// TIA Portal V20 export
FUNCTION_BLOCK "FB_Temperature"   // FB490, SCL
{ S7_Optimized_Access := 'TRUE' }
// stored: AutoNumber false, MemoryReserve 100, SetENOAutomatically false
   VAR
      sPIDRestart : Bool;
      sPIDHoldI : Bool;
      sXAxisWarning : Real := 50.0;
      sPIDClimOut : Real;
      sP : Real := -100.0;
      sI : Time := T#10D;
      sD : Time := T#12S;
      sTimeOutFlowChiller : TON_TIME;
      sTimeOutLevelChiller { S7_SetPoint := 'True'} : TON_TIME;
      sTimeOutChillerGood : TON_TIME;
      sTimeOutCooling : TON_TIME;
      sTemperature_X_PT1000 { S7_SetPoint := 'True'} : "FB_AnalogInputThreshold";
      sTemperature_Y_PT1000 { S7_SetPoint := 'True'} : "FB_AnalogInputThreshold";
      sAmbiantTemperature { S7_SetPoint := 'True'} : "FB_AnalogInputThreshold";
      sMachineTemperature { S7_SetPoint := 'True'} : "FB_AnalogInputThreshold";
      sCabinetTemperatureMeasure { S7_SetPoint := 'True'} : "FB_AnalogInputThreshold";
      sColdWaterTemperatureInput { S7_SetPoint := 'True'} : "FB_AnalogInputThreshold";
      sColdWaterTemperatureOutput { S7_SetPoint := 'True'} : "FB_AnalogInputThreshold";
      sTemperatureCooling { S7_SetPoint := 'True'} : "FB_AnalogInputThreshold";
   END_VAR
   VAR_TEMP
      tSetPointCheck : Real;
      tDataAction : "AnalogInAction_DT";
   END_VAR
   VAR CONSTANT
      ALARM_PTC : Real := 110.0;
      TIME_OUT_COOLING : Time := T#5S;
   END_VAR
BEGIN
   REGION Description header 
       //==================================================================================
       // POSALUX Swiss SA / (C) Copyright 2024
       //----------------------------------------------------------------------------------
       // Title: Temperatures management
       // Comment/Function: 
       //
       // Author: Gowsigan SRITHARAN
       // Engineering: TIA Portal v17
       //----------------------------------------------------------------------------------
       // Change log table:
       // Version  | Date     | Expert in charge | Changes applied
       // ---------|----------|------------------|------------------------------------
       // 00.00.01 | 20241120 | GSR              | First released version
       // ==================================================================================
   END_REGION

   REGION Ambiant temperature (externe)  
       #sAmbiantTemperature(iActualValue := "DB_AnalogInputs".sAmbiantTemperature.sSWRealValue,
                            iStartDelay := TRUE,
                            ioAlarmMin := "LBP_AlarmMsgs".UserA[06].A70UUxx[04],
                            ioWarningMin := "LBP_AlarmMsgs".UserA[07].A70UUxx[04],
                            ioWarningMax := "LBP_AlarmMsgs".UserA[07].A70UUxx[05],
                            ioAlarmMax := "LBP_AlarmMsgs".UserA[06].A70UUxx[05],
                            oDataAction => "DB_AnalogInputAction".Ambiant_Temperature,
                            iDataPLC := "DB_AnalogInputDataPLC".Ambiant_Temperature,
                            iDataHMI := "DB_AnalogInputDataHMI".Ambiant_Temperature);
   END_REGION

   REGION Water input  
       #sColdWaterTemperatureInput(iActualValue := "DB_AnalogInputs".sCold_WaterTemperatureInput.sSWRealValue,
                                   iStartDelay := TRUE,
                                   ioAlarmMin := "LBP_AlarmMsgs".UserA[06].A70UUxx[08],
                                   ioWarningMin := "LBP_AlarmMsgs".UserA[07].A70UUxx[08],
                                   ioWarningMax := "LBP_AlarmMsgs".UserA[07].A70UUxx[09],
                                   ioAlarmMax := "LBP_AlarmMsgs".UserA[06].A70UUxx[09],
                                   oDataAction => "DB_AnalogInputAction".Cold_Water_Temperature_Input,
                                   iDataPLC := "DB_AnalogInputDataPLC".Cold_Water_Temperature_Input,
                                   iDataHMI := "DB_AnalogInputDataHMI".Cold_Water_Temperature_Input);
   END_REGION

   REGION Cooling On
       "DB_DigitalOutputs".sCoolingStart.sSWStatus := "DB_PowerOn".sMachineReadySoft;
   END_REGION ;

   REGION Cooling alarm
       #sTimeOutCooling(IN := "DB_PowerOn".sTimeMachineReadyDelay.Q AND NOT "DB_DigitalInputs".sCoolingOK.sSWStatus,
                        PT := #TIME_OUT_COOLING,
                        Q => "LBP_AlarmMsgs".UserA[4].A70UUxx[10]);
   END_REGION

   REGION Water output   
       #sColdWaterTemperatureOutput(iActualValue := "DB_AnalogInputs".sCold_WaterTemperatureOutput.sSWRealValue,
                                    iStartDelay := TRUE,
                                    ioAlarmMin := "LBP_AlarmMsgs".UserA[06].A70UUxx[10],
                                    ioWarningMin := "LBP_AlarmMsgs".UserA[07].A70UUxx[10],
                                    ioWarningMax := "LBP_AlarmMsgs".UserA[07].A70UUxx[11],
                                    ioAlarmMax := "LBP_AlarmMsgs".UserA[06].A70UUxx[11],
                                    oDataAction => "DB_AnalogInputAction".Cold_Water_Temperature_Output,
                                    iDataPLC := "DB_AnalogInputDataPLC".Cold_Water_Temperature_Output,
                                    iDataHMI := "DB_AnalogInputDataHMI".Cold_Water_Temperature_Output);
   END_REGION

   REGION X Axis temperature check
       #sTemperature_X_PT1000(iActualValue := "DB_AnalogInputs".sX_AxisTemperaturePT1000.sSWRealValue,
                              iStartDelay := TRUE,
                              ioAlarmMin := "LBP_AlarmMsgs".UserA[06].A70UUxx[00],
                              ioWarningMin := "LBP_AlarmMsgs".UserA[07].A70UUxx[00],
                              ioWarningMax := "LBP_AlarmMsgs".UserA[07].A70UUxx[01],
                              ioAlarmMax := "LBP_AlarmMsgs".UserA[06].A70UUxx[01],
                              oDataAction => "DB_AnalogInputAction".X_Axis_Temperature_PT1000,
                              iDataPLC := "DB_AnalogInputDataPLC".X_Axis_Temperature_PT1000,
                              iDataHMI := "DB_AnalogInputDataHMI".X_Axis_Temperature_PT1000);

       // Temperature_X_PTC
       // PTC used as a temperature threshold rather than a measurement
       IF "DB_AnalogInputs".sX_AxisTemperaturePTC.iValueHW.%X0 OR "DB_AnalogInputs".sX_AxisTemperaturePTC.iValueHW.%X2 THEN
           "LBP_AlarmMsgs".UserA[06].A70UUxx[23] := TRUE;
       END_IF;
   END_REGION

   REGION Y Axis temperature check
       #sTemperature_Y_PT1000(iActualValue := "DB_AnalogInputs".sY_AxisTemperaturePT1000.sSWRealValue,
                              iStartDelay := TRUE,
                              ioAlarmMin := "LBP_AlarmMsgs".UserA[06].A70UUxx[02],
                              ioWarningMin := "LBP_AlarmMsgs".UserA[07].A70UUxx[02],
                              ioWarningMax := "LBP_AlarmMsgs".UserA[07].A70UUxx[03],
                              ioAlarmMax := "LBP_AlarmMsgs".UserA[06].A70UUxx[03],
                              oDataAction => "DB_AnalogInputAction".Y_Axis_Temperature_PT1000,
                              iDataPLC := "DB_AnalogInputDataPLC".Y_Axis_Temperature_PT1000,
                              iDataHMI := "DB_AnalogInputDataHMI".Y_Axis_Temperature_PT1000);

       // Temperature_Y_PTC
       // PTC used as a temperature threshold rather than a measurement
       IF "DB_AnalogInputs".sY_AxisTemperaturePTC.iValueHW.%X0 OR "DB_AnalogInputs".sY_AxisTemperaturePTC.iValueHW.%X2 THEN
           "LBP_AlarmMsgs".UserA[06].A70UUxx[25] := TRUE;
       END_IF;
   END_REGION

   REGION Electrical Cabinet
       #sCabinetTemperatureMeasure(iActualValue := "DB_AnalogInputs".sCabinetTemperature.sSWRealValue,
                                   iStartDelay := TRUE,
                                   ioAlarmMin := "LBP_AlarmMsgs".UserA[06].A70UUxx[52],
                                   ioWarningMin := "LBP_AlarmMsgs".UserA[07].A70UUxx[52],
                                   ioWarningMax := "LBP_AlarmMsgs".UserA[07].A70UUxx[53],
                                   ioAlarmMax := "LBP_AlarmMsgs".UserA[06].A70UUxx[53],
                                   oDataAction => "DB_AnalogInputAction".Cabinet_Temperature,
                                   iDataPLC := "DB_AnalogInputDataPLC".Cabinet_Temperature,
                                   iDataHMI := "DB_AnalogInputDataHMI".Cabinet_Temperature);

       IF "DB_DigitalInputs".sCabinetTemperatureCtrl.sSWStatus THEN
            "LBP_AlarmMsgs".UserA[0].A70UUxx[4] := TRUE;
        END_IF;
    END_REGION

    REGION Machine management temperature (interieur)
        #sMachineTemperature(iActualValue := "DB_AnalogInputs".sMachineTemperature.sSWRealValue,
                             iStartDelay := TRUE,
                             ioAlarmMin := "LBP_AlarmMsgs".UserA[06].A70UUxx[06],
                             ioWarningMin := "LBP_AlarmMsgs".UserA[07].A70UUxx[06],
                             ioWarningMax := "LBP_AlarmMsgs".UserA[07].A70UUxx[07],
                             ioAlarmMax := "LBP_AlarmMsgs".UserA[06].A70UUxx[07],
                             oDataAction => "DB_AnalogInputAction".Machine_Temperature,
                             iDataPLC := "DB_AnalogInputDataPLC".Machine_Temperature,
                             iDataHMI := "DB_AnalogInputDataHMI".Machine_Temperature);

        REGION Machine ventilator
            // Ventilator setpoint (from HMI) Forcing value under 0% OR over 100%
            IF "DB_HMISetting".CoolingVentilatorSetpoint < 0.0 THEN
                "DB_HMISetting".CoolingVentilatorSetpoint := 0.0;
            ELSIF "DB_HMISetting".CoolingVentilatorSetpoint > 100.0 THEN
                "DB_HMISetting".CoolingVentilatorSetpoint := 100.0;
            END_IF;

            IF "DB_DigitalOutputs".sXY_AxisPowerContactor.sSWStatus OR
                "DB_DigitalOutputs".sAxis2_PowerContactor.sSWStatus OR
                "DB_DigitalOutputs".sBus60V_PowerContactor.sSWStatus THEN
                "DB_AnalogOutputs".sVentilatorSetPoint.sSWRealValue := "DB_HMISetting".CoolingVentilatorSetpoint;
            ELSE
                "DB_AnalogOutputs".sVentilatorSetPoint.sSWRealValue := 0.0;
            END_IF;
        END_REGION

        REGION Check setpoint temperature machine
            #sTemperatureCooling(iActualValue := "DB_AnalogInputs".sClimTemperature.sSWRealValue,
                                 iStartDelay := TRUE,
                                 ioAlarmMin := "LBP_AlarmMsgs".UserA[06].A70UUxx[54],
                                 ioWarningMin := "LBP_AlarmMsgs".UserA[07].A70UUxx[54],
                                 ioWarningMax := "LBP_AlarmMsgs".UserA[07].A70UUxx[55],
                                 ioAlarmMax := "LBP_AlarmMsgs".UserA[06].A70UUxx[55],
                                 oDataAction => #tDataAction,
                                 iDataPLC := "DB_AnalogInputDataPLC".Clim_Temperature,
                                 iDataHMI := "DB_AnalogInputDataHMI".Clim_Temperature);
        END_REGION

        // REGION Machine temperature cooling PID WFA Déplacé dans OB30
        //     "CONT_C_Clim_DB"(COM_RST := #sPIDRestart,
        //                      MAN_ON := FALSE,
        //                      P_SEL := TRUE,
        //                      I_SEL := TRUE,
        //                      INT_HOLD := #sPIDHoldI,
        //                      D_SEL := TRUE,
        //                      CYCLE := T#1s,
        //                      SP_INT := "DB_HMISetting".TemperatureCoolingSetpoint,
        //                      PV_IN := "DB_AnalogInputs".sClimTemperature.sSWRealValue,
        //                      GAIN := #sP,
        //                      TI := #sI,
        //                      TD := #sD,
        //                      DEADB_W := 0.1,
        //                      LMN_HLM := 100,
        //                      LMN_LLM := 0,
        //                      LMN => "DB_AnalogOutputs".sPropValveClimSetPoint.sSWRealValue);
        // END_REGION
    END_REGION
END_FUNCTION_BLOCK
